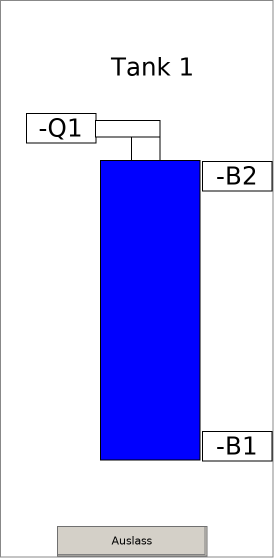
VISUALIZATION TankFuellAnlage  // 274x558
    Rectangle (131,120 29x305), colour toggle: DIO.Q1
    Rectangle (100,160 100x300)
    Rectangle (100,160 100x300)
        p2773130477: MAIN.Simulation.uiFuellstandTank1
    Label (105,52 95x30), "Tank 1"
    Button (57,526 150x30), "Auslass"
        tap MAIN.Simulation.xAuslass1
    Rectangle (202,161 70x30), "-B2", colour toggle: VISU.B2
    Rectangle (202,431 70x30), "-B1", colour toggle: VISU.B1
    Rectangle (26,113 70x30), "-Q1", colour toggle: DIO.Q1
    Rectangle (95,120 65x17), colour toggle: DIO.Q1
    Rectangle (86,186 29x301), colour toggle: DIO.Q1
END_VISUALIZATION

(* stored: Version 1.1.0.1, ProductVersion 3.1.4022.6
   Visu TankFuellAnlage: Id {116ef40b-496c-489a-a025-1af3552c8f1e} *)
